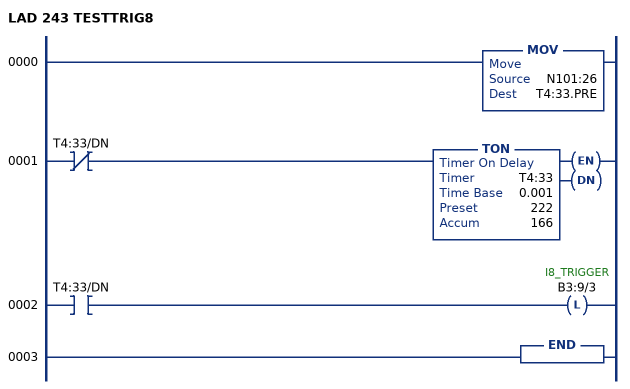
% Rung: 0 %
SOR MOV N101:26 T4:33.PRE EOR
%   N101:26  I8_TRIGTIME %
% Rung: 1 %
SOR XIO T4:33/DN TON T4:33 0.001 222 166 EOR
% Rung: 2 %
SOR XIC T4:33/DN OTL B3:9/3 EOR
%   B3:9/3  I8_TRIGGER %
% Rung: 3 %
SOR END EOR

LADDER 244 "PACKAGER"    % normal %
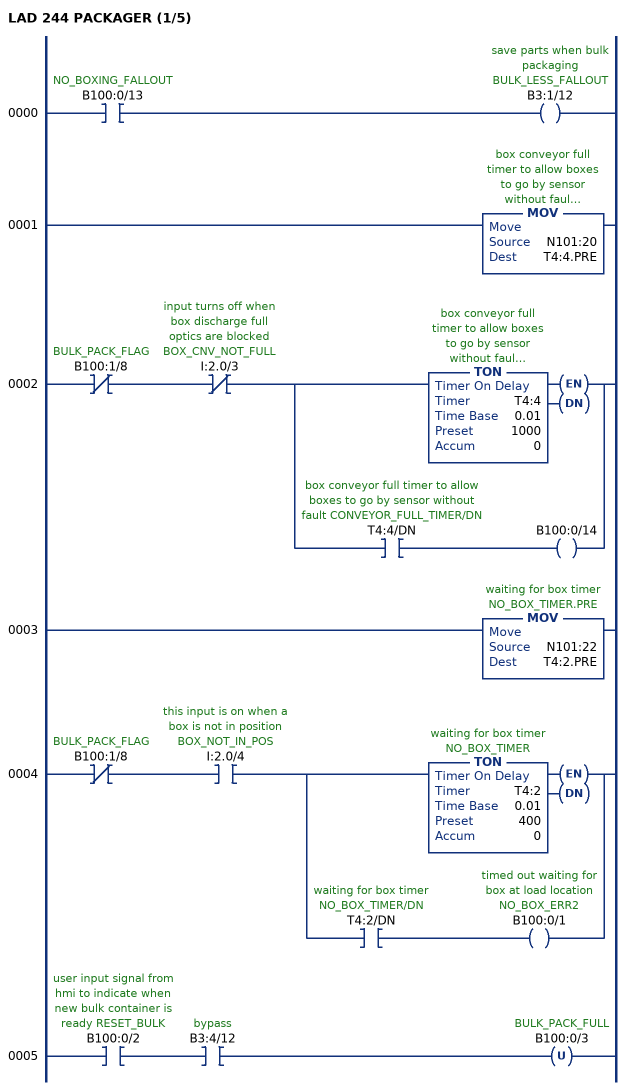
% Rung: 0 %
SOR XIC B100:0/13 OTE B3:1/12 EOR
%   B100:0/13  NO_BOXING_FALLOUT %
%   B3:1/12  BULK_LESS_FALLOUT  "save parts when bulk packaging" %
% Rung: 1 %
SOR MOV N101:20 T4:4.PRE EOR
%   N101:20  CONV_FULL_TIME_LIMIT  "time to allow box to pass box conveyor full sensor without fault" %
%   T4:4  CONVEYOR_FULL_TIMER  "box conveyor full timer to allow boxes to go by sensor without fault" %
% Rung: 2 %
SOR XIO B100:1/8 XIO I:2.0/3 BST TON T4:4 0.01 1000 0 NXB XIC T4:4/DN OTE B100:0/14 BND EOR
%   B100:1/8  BULK_PACK_FLAG %
%   I:2.0/3  BOX_CNV_NOT_FULL  "input turns off when box discharge full optics are blocked" %
%   T4:4  CONVEYOR_FULL_TIMER  "box conveyor full timer to allow boxes to go by sensor without fault" %
% Rung: 3 %
SOR MOV N101:22 T4:2.PRE EOR
%   N101:22  BOX_WAIT_TIME_LIMIT  "the time until waiting for box message in hmi (fault)" %
%   T4:2  NO_BOX_TIMER  "waiting for box timer" %
% Rung: 4 %
SOR XIO B100:1/8 XIC I:2.0/4 BST TON T4:2 0.01 400 0 NXB XIC T4:2/DN OTE B100:0/1 BND EOR
%   B100:1/8  BULK_PACK_FLAG %
%   I:2.0/4  BOX_NOT_IN_POS  "this input is on when a box is not in position" %
%   T4:2  NO_BOX_TIMER  "waiting for box timer" %
%   B100:0/1  NO_BOX_ERR2  "timed out waiting for box at load location" %
% Rung: 5 %
SOR XIC B100:0/2 XIC B3:4/12 OTU B100:0/3 EOR
%   B100:0/2  RESET_BULK  "user input signal from hmi to indicate when new bulk container is ready" %
%   B3:4/12  "bypass" %
%   B100:0/3  BULK_PACK_FULL %

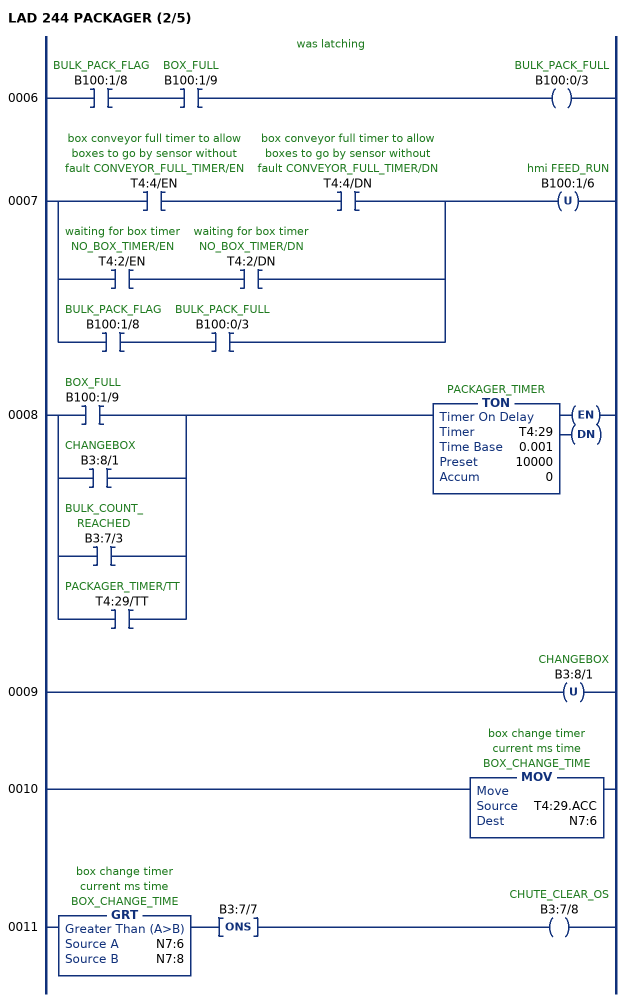
% Rung: 6 %
% was latching %
SOR XIC B100:1/8 XIC B100:1/9 OTE B100:0/3 EOR
%   B100:1/8  BULK_PACK_FLAG %
%   B100:1/9  BOX_FULL %
%   B100:0/3  BULK_PACK_FULL %
% Rung: 7 %
SOR BST XIC T4:4/EN XIC T4:4/DN NXB XIC T4:2/EN XIC T4:2/DN NXB XIC B100:1/8 XIC B100:0/3 BND OTU B100:1/6 EOR
%   T4:4  CONVEYOR_FULL_TIMER  "box conveyor full timer to allow boxes to go by sensor without fault" %
%   T4:2  NO_BOX_TIMER  "waiting for box timer" %
%   B100:1/8  BULK_PACK_FLAG %
%   B100:0/3  BULK_PACK_FULL %
%   B100:1/6  FEED_RUN  "hmi" %
% Rung: 8 %
SOR BST XIC B100:1/9 NXB XIC B3:8/1 NXB XIC B3:7/3 NXB XIC T4:29/TT BND TON T4:29 0.001 10000 0 EOR
%   B100:1/9  BOX_FULL %
%   B3:8/1  CHANGEBOX %
%   B3:7/3  BULK_COUNT_REACHED %
%   T4:29  PACKAGER_TIMER %
% Rung: 9 %
SOR OTU B3:8/1 EOR
%   B3:8/1  CHANGEBOX %
% Rung: 10 %
SOR MOV T4:29.ACC N7:6 EOR
%   T4:29  PACKAGER_TIMER %
%   N7:6  BOX_CHANGE_TIME  "box change timer current ms time" %
% Rung: 11 %
SOR GRT N7:6 N7:8 ONS B3:7/7 OTE B3:7/8 EOR
%   N7:6  BOX_CHANGE_TIME  "box change timer current ms time" %
%   N7:8  CHUTE_CLEAR_TIME %
%   B3:7/8  CHUTE_CLEAR_OS %

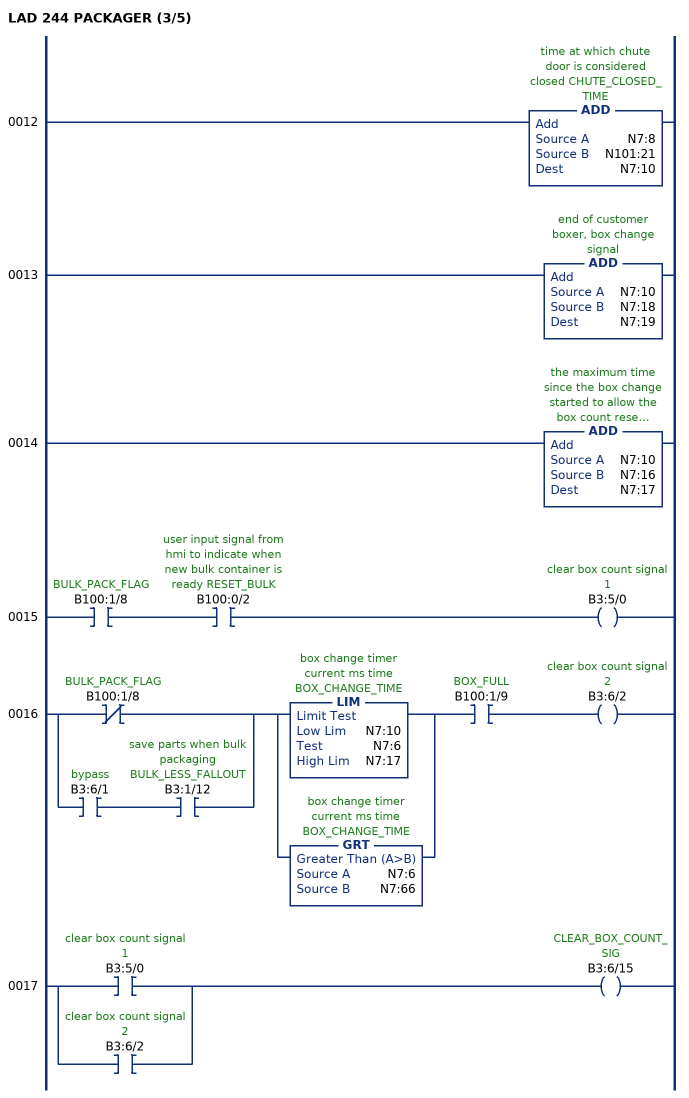
% Rung: 12 %
SOR ADD N7:8 N101:21 N7:10 EOR
%   N7:8  CHUTE_CLEAR_TIME %
%   N101:21  CHUTE_CLOSE_TIME  "ms time required to close chute" %
%   N7:10  CHUTE_CLOSED_TIME  "time at which chute door is considered closed" %
% Rung: 13 %
SOR ADD N7:10 N7:18 N7:19 EOR
%   N7:10  CHUTE_CLOSED_TIME  "time at which chute door is considered closed" %
%   N7:18  CHANGE_BOX_SIG_TIME  "customer boxer change box signal time" %
%   N7:19  "end of customer boxer, box change signal" %
% Rung: 14 %
SOR ADD N7:10 N7:16 N7:17 EOR
%   N7:10  CHUTE_CLOSED_TIME  "time at which chute door is considered closed" %
%   N7:16  RESET_COUNT_SIG_TIME  "maximum length of time to hold box count reset signal on" %
%   N7:17  "the maximum time since the box change started to allow the box count reset signal" %
% Rung: 15 %
SOR XIC B100:1/8 XIC B100:0/2 OTE B3:5/0 EOR
%   B100:1/8  BULK_PACK_FLAG %
%   B100:0/2  RESET_BULK  "user input signal from hmi to indicate when new bulk container is ready" %
%   B3:5/0  "clear box count signal 1" %
% Rung: 16 %
SOR BST XIO B100:1/8 NXB XIC B3:6/1 XIC B3:1/12 BND BST LIM N7:10 N7:6 N7:17 NXB GRT N7:6 N7:66 BND XIC B100:1/9 OTE B3:6/2 EOR
%   B100:1/8  BULK_PACK_FLAG %
%   B3:6/1  "bypass" %
%   B3:1/12  BULK_LESS_FALLOUT  "save parts when bulk packaging" %
%   N7:10  CHUTE_CLOSED_TIME  "time at which chute door is considered closed" %
%   N7:6  BOX_CHANGE_TIME  "box change timer current ms time" %
%   N7:17  "the maximum time since the box change started to allow the box count reset signal" %
%   B100:1/9  BOX_FULL %
%   B3:6/2  "clear box count signal 2" %
% Rung: 17 %
SOR BST XIC B3:5/0 NXB XIC B3:6/2 BND OTE B3:6/15 EOR
%   B3:5/0  "clear box count signal 1" %
%   B3:6/2  "clear box count signal 2" %
%   B3:6/15  CLEAR_BOX_COUNT_SIG %

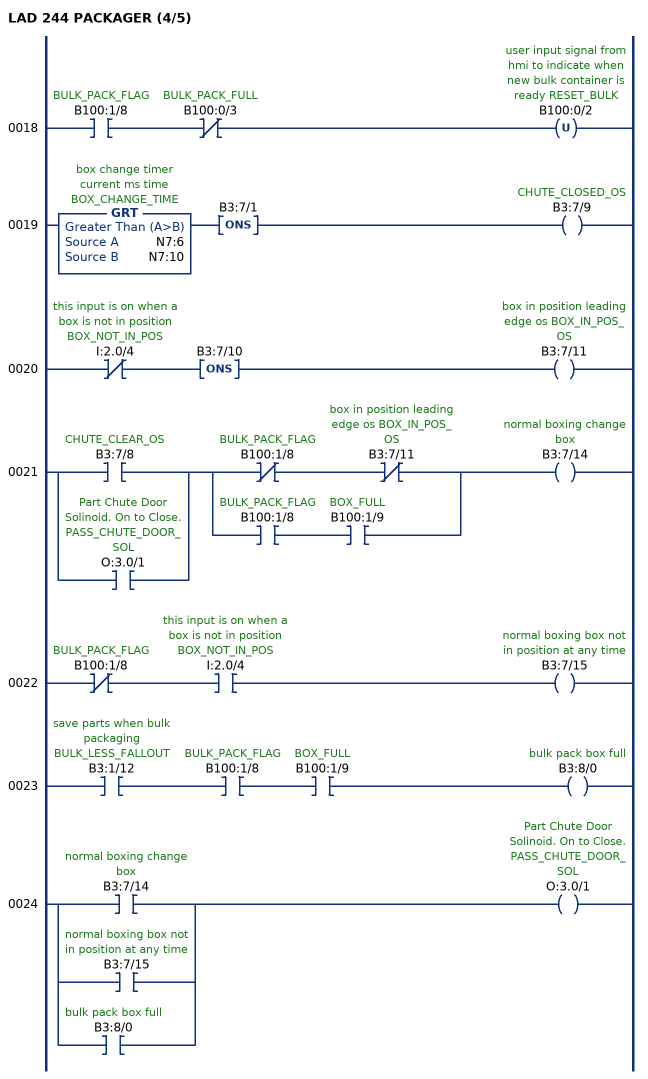
% Rung: 18 %
SOR XIC B100:1/8 XIO B100:0/3 OTU B100:0/2 EOR
%   B100:1/8  BULK_PACK_FLAG %
%   B100:0/3  BULK_PACK_FULL %
%   B100:0/2  RESET_BULK  "user input signal from hmi to indicate when new bulk container is ready" %
% Rung: 19 %
SOR GRT N7:6 N7:10 ONS B3:7/1 OTE B3:7/9 EOR
%   N7:6  BOX_CHANGE_TIME  "box change timer current ms time" %
%   N7:10  CHUTE_CLOSED_TIME  "time at which chute door is considered closed" %
%   B3:7/9  CHUTE_CLOSED_OS %
% Rung: 20 %
SOR XIO I:2.0/4 ONS B3:7/10 OTE B3:7/11 EOR
%   I:2.0/4  BOX_NOT_IN_POS  "this input is on when a box is not in position" %
%   B3:7/11  BOX_IN_POS_OS  "box in position leading edge os" %
% Rung: 21 %
SOR BST XIC B3:7/8 NXB XIC O:3.0/1 BND BST XIO B100:1/8 XIO B3:7/11 NXB XIC B100:1/8 XIC B100:1/9 BND OTE B3:7/14 EOR
%   B3:7/8  CHUTE_CLEAR_OS %
%   O:3.0/1  PASS_CHUTE_DOOR_SOL  "Part Chute Door Solinoid. On to Close." %
%   B100:1/8  BULK_PACK_FLAG %
%   B3:7/11  BOX_IN_POS_OS  "box in position leading edge os" %
%   B100:1/9  BOX_FULL %
%   B3:7/14  "normal boxing change box" %
% Rung: 22 %
SOR XIO B100:1/8 XIC I:2.0/4 OTE B3:7/15 EOR
%   B100:1/8  BULK_PACK_FLAG %
%   I:2.0/4  BOX_NOT_IN_POS  "this input is on when a box is not in position" %
%   B3:7/15  "normal boxing box not in position at any time" %
% Rung: 23 %
SOR XIC B3:1/12 XIC B100:1/8 XIC B100:1/9 OTE B3:8/0 EOR
%   B3:1/12  BULK_LESS_FALLOUT  "save parts when bulk packaging" %
%   B100:1/8  BULK_PACK_FLAG %
%   B100:1/9  BOX_FULL %
%   B3:8/0  "bulk pack box full" %
% Rung: 24 %
SOR BST XIC B3:7/14 NXB XIC B3:7/15 NXB XIC B3:8/0 BND OTE O:3.0/1 EOR
%   B3:7/14  "normal boxing change box" %
%   B3:7/15  "normal boxing box not in position at any time" %
%   B3:8/0  "bulk pack box full" %
%   O:3.0/1  PASS_CHUTE_DOOR_SOL  "Part Chute Door Solinoid. On to Close." %

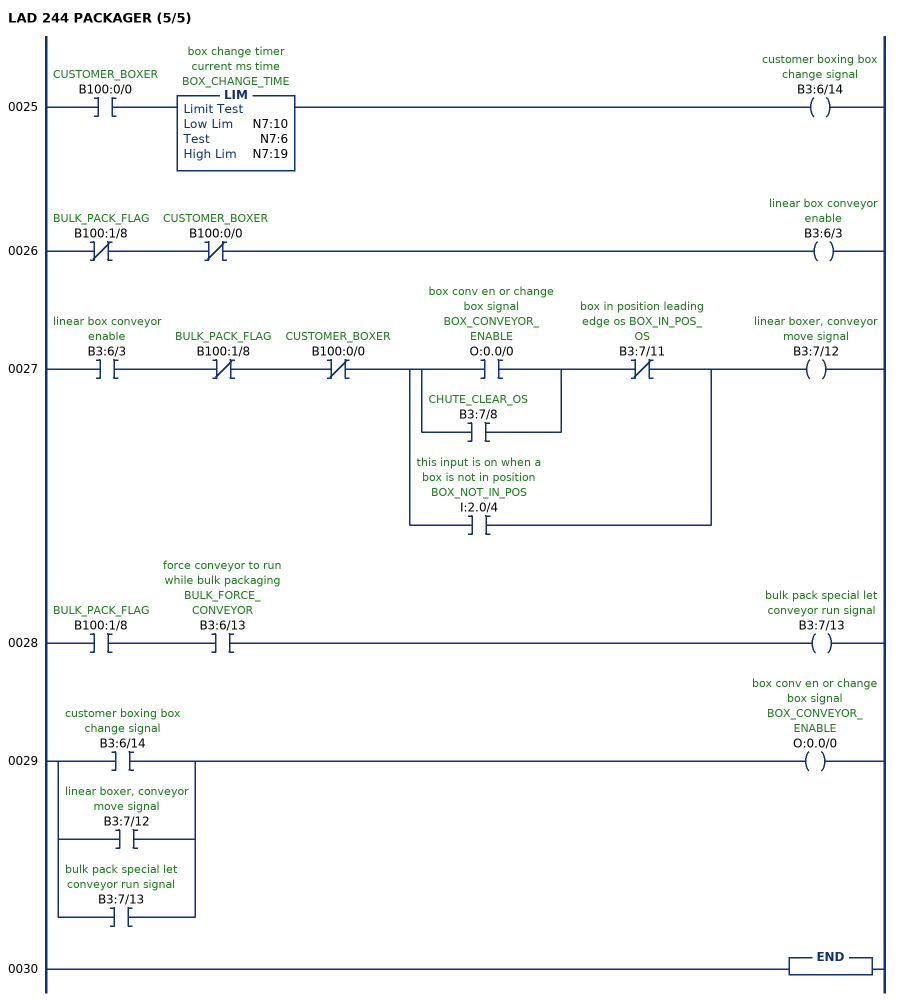
% Rung: 25 %
SOR XIC B100:0/0 LIM N7:10 N7:6 N7:19 OTE B3:6/14 EOR
%   B100:0/0  CUSTOMER_BOXER %
%   N7:10  CHUTE_CLOSED_TIME  "time at which chute door is considered closed" %
%   N7:6  BOX_CHANGE_TIME  "box change timer current ms time" %
%   N7:19  "end of customer boxer, box change signal" %
%   B3:6/14  "customer boxing box change signal" %
% Rung: 26 %
SOR XIO B100:1/8 XIO B100:0/0 OTE B3:6/3 EOR
%   B100:1/8  BULK_PACK_FLAG %
%   B100:0/0  CUSTOMER_BOXER %
%   B3:6/3  "linear box conveyor enable" %
% Rung: 27 %
SOR XIC B3:6/3 XIO B100:1/8 XIO B100:0/0 BST BST XIC O:0.0/0 NXB XIC B3:7/8 BND XIO B3:7/11 NXB XIC I:2.0/4 BND OTE B3:7/12 EOR
%   B3:6/3  "linear box conveyor enable" %
%   B100:1/8  BULK_PACK_FLAG %
%   B100:0/0  CUSTOMER_BOXER %
%   O:0.0/0  BOX_CONVEYOR_ENABLE  "box conv en or change box signal" %
%   B3:7/8  CHUTE_CLEAR_OS %
%   B3:7/11  BOX_IN_POS_OS  "box in position leading edge os" %
%   I:2.0/4  BOX_NOT_IN_POS  "this input is on when a box is not in position" %
%   B3:7/12  "linear boxer, conveyor move signal" %
% Rung: 28 %
SOR XIC B100:1/8 XIC B3:6/13 OTE B3:7/13 EOR
%   B100:1/8  BULK_PACK_FLAG %
%   B3:6/13  BULK_FORCE_CONVEYOR  "force conveyor to run while bulk packaging" %
%   B3:7/13  "bulk pack special let conveyor run signal" %
% Rung: 29 %
SOR BST XIC B3:6/14 NXB XIC B3:7/12 NXB XIC B3:7/13 BND OTE O:0.0/0 EOR
%   B3:6/14  "customer boxing box change signal" %
%   B3:7/12  "linear boxer, conveyor move signal" %
%   B3:7/13  "bulk pack special let conveyor run signal" %
%   O:0.0/0  BOX_CONVEYOR_ENABLE  "box conv en or change box signal" %
% Rung: 30 %
SOR END EOR

LADDER 245 "NO PACKAGE"
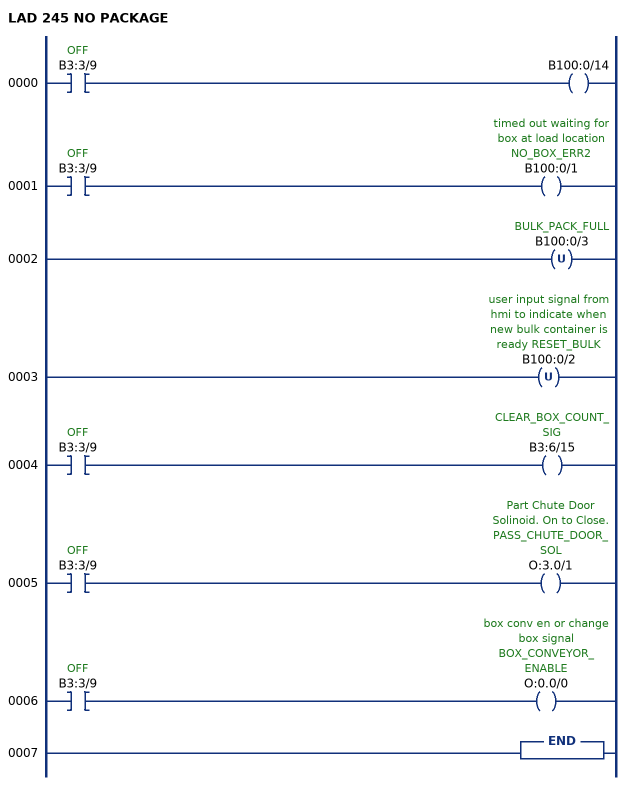
% Rung: 0 %
SOR XIC B3:3/9 OTE B100:0/14 EOR
%   B3:3/9  OFF %
% Rung: 1 %
SOR XIC B3:3/9 OTE B100:0/1 EOR
%   B3:3/9  OFF %
%   B100:0/1  NO_BOX_ERR2  "timed out waiting for box at load location" %
% Rung: 2 %
SOR OTU B100:0/3 EOR
%   B100:0/3  BULK_PACK_FULL %
% Rung: 3 %
SOR OTU B100:0/2 EOR
%   B100:0/2  RESET_BULK  "user input signal from hmi to indicate when new bulk container is ready" %
% Rung: 4 %
SOR XIC B3:3/9 OTE B3:6/15 EOR
%   B3:3/9  OFF %
%   B3:6/15  CLEAR_BOX_COUNT_SIG %
% Rung: 5 %
SOR XIC B3:3/9 OTE O:3.0/1 EOR
%   B3:3/9  OFF %
%   O:3.0/1  PASS_CHUTE_DOOR_SOL  "Part Chute Door Solinoid. On to Close." %
% Rung: 6 %
SOR XIC B3:3/9 OTE O:0.0/0 EOR
%   B3:3/9  OFF %
%   O:0.0/0  BOX_CONVEYOR_ENABLE  "box conv en or change box signal" %
% Rung: 7 %
SOR END EOR

LADDER 246 "RATE1"
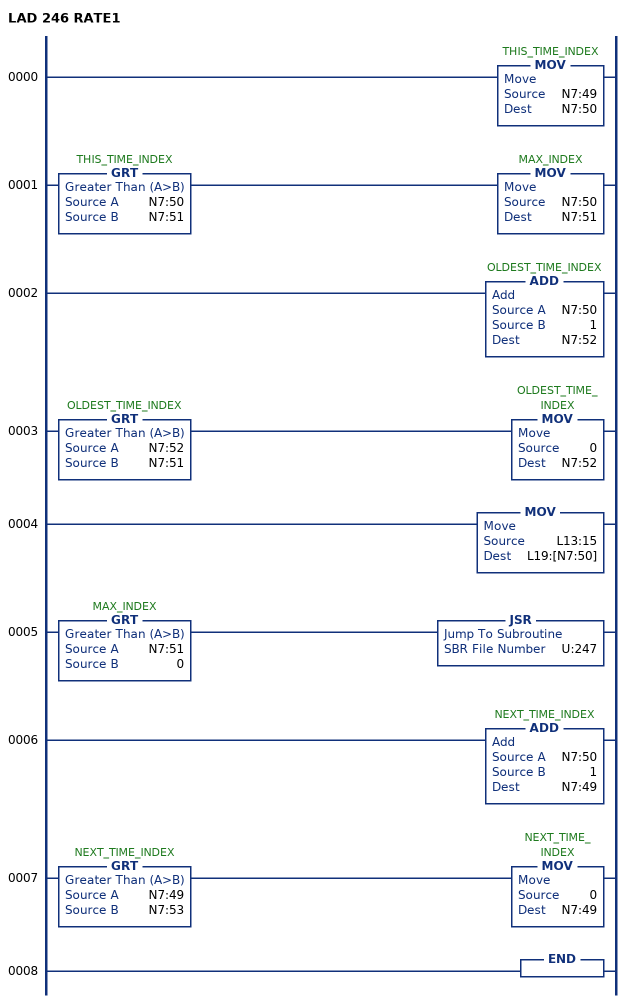
% Rung: 0 %
SOR MOV N7:49 N7:50 EOR
%   N7:49  NEXT_TIME_INDEX %
%   N7:50  THIS_TIME_INDEX %
% Rung: 1 %
SOR GRT N7:50 N7:51 MOV N7:50 N7:51 EOR
%   N7:50  THIS_TIME_INDEX %
%   N7:51  MAX_INDEX %
% Rung: 2 %
SOR ADD N7:50 1 N7:52 EOR
%   N7:50  THIS_TIME_INDEX %
%   N7:52  OLDEST_TIME_INDEX %
% Rung: 3 %
SOR GRT N7:52 N7:51 MOV 0 N7:52 EOR
%   N7:52  OLDEST_TIME_INDEX %
%   N7:51  MAX_INDEX %
% Rung: 4 %
SOR MOV L13:15 L19:[N7:50] EOR
%   L13:15  THE_TIME %
%   N7:50  THIS_TIME_INDEX %
% Rung: 5 %
SOR GRT N7:51 0 JSR U:247 EOR
%   N7:51  MAX_INDEX %
% Rung: 6 %
SOR ADD N7:50 1 N7:49 EOR
%   N7:50  THIS_TIME_INDEX %
%   N7:49  NEXT_TIME_INDEX %
% Rung: 7 %
SOR GRT N7:49 N7:53 MOV 0 N7:49 EOR
%   N7:49  NEXT_TIME_INDEX %
%   N7:53  UPPER_INDEX_LIMIT %
% Rung: 8 %
SOR END EOR

LADDER 247 "RATE2"
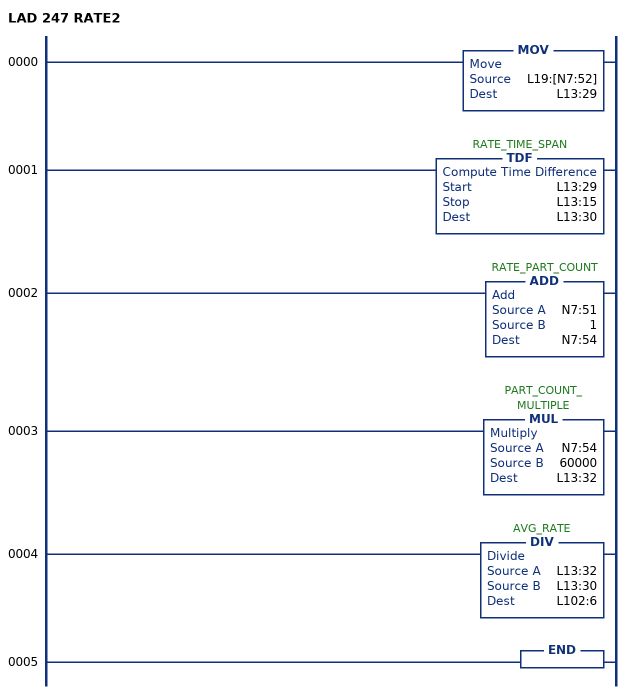
% Rung: 0 %
SOR MOV L19:[N7:52] L13:29 EOR
%   N7:52  OLDEST_TIME_INDEX %
% Rung: 1 %
SOR TDF L13:29 L13:15 L13:30 EOR
%   L13:15  THE_TIME %
%   L13:30  RATE_TIME_SPAN %
% Rung: 2 %
SOR ADD N7:51 1 N7:54 EOR
%   N7:51  MAX_INDEX %
%   N7:54  RATE_PART_COUNT %
% Rung: 3 %
SOR MUL N7:54 60000 L13:32 EOR
%   N7:54  RATE_PART_COUNT %
%   L13:32  PART_COUNT_MULTIPLE %
% Rung: 4 %
SOR DIV L13:32 L13:30 L102:6 EOR
%   L13:32  PART_COUNT_MULTIPLE %
%   L13:30  RATE_TIME_SPAN %
%   L102:6  AVG_RATE %
% Rung: 5 %
SOR END EOR

LADDER 248 "RESET RATE"
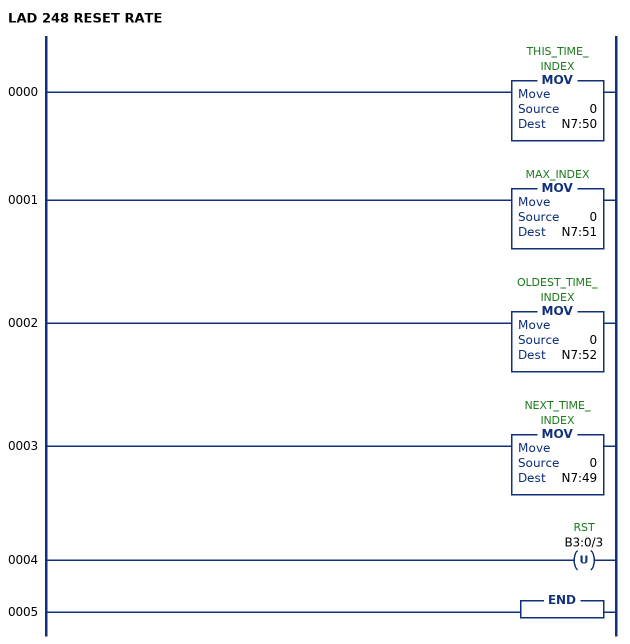
% Rung: 0 %
SOR MOV 0 N7:50 EOR
%   N7:50  THIS_TIME_INDEX %
% Rung: 1 %
SOR MOV 0 N7:51 EOR
%   N7:51  MAX_INDEX %
% Rung: 2 %
SOR MOV 0 N7:52 EOR
%   N7:52  OLDEST_TIME_INDEX %
% Rung: 3 %
SOR MOV 0 N7:49 EOR
%   N7:49  NEXT_TIME_INDEX %
% Rung: 4 %
SOR OTU B3:0/3 EOR
%   B3:0/3  RST %
% Rung: 5 %
SOR END EOR

LADDER 249 "NP STOP"    % stop on no good %
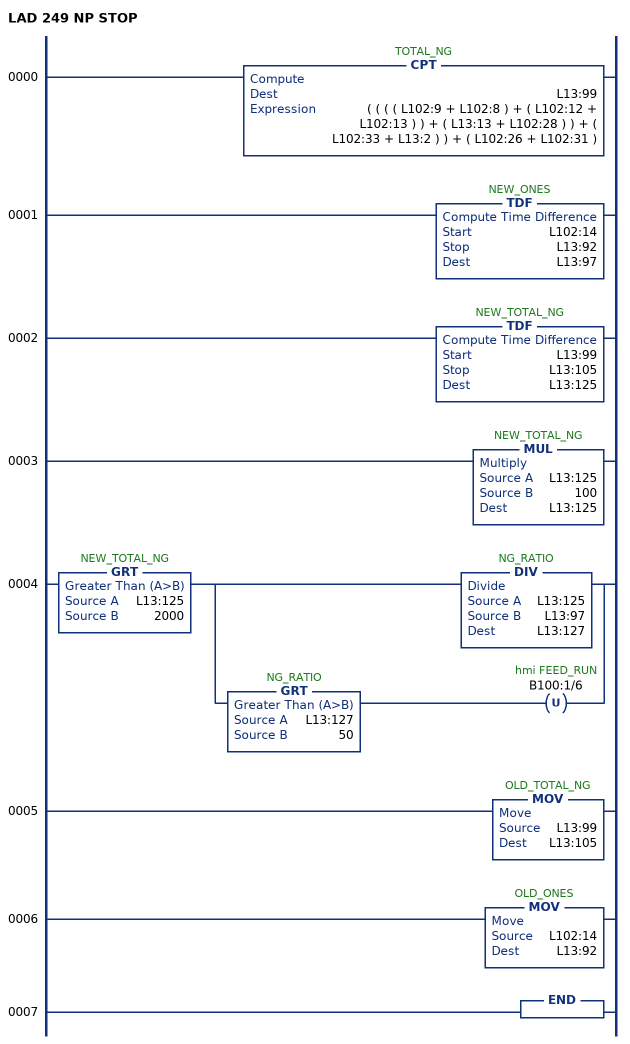
% Rung: 0 %
SOR CPT L13:99 " ( ( ( ( L102:9 + L102:8 ) + ( L102:12 + L102:13 ) ) + ( L13:13 + L102:28 ) ) + ( L102:33 + L13:2 ) ) + ( L102:26 + L102:31 ) " EOR
%   L13:99  TOTAL_NG %
%   L102:9  "too wide bottom" %
%   L102:8  "too close bottom" %
%   L102:12  "too close top count" %
%   L102:13  "too wide top count" %
%   L102:28  I1_I5_SKIPPEDCOUNT %
%   L102:33  I2_I6_SKIPPEDCOUNT %
%   L102:26  I1_I5_FAIL_COUNT %
%   L102:31  I2_I6_FAIL_COUNT %
% Rung: 1 %
SOR TDF L102:14 L13:92 L13:97 EOR
%   L102:14  ONES %
%   L13:92  OLD_ONES %
%   L13:97  NEW_ONES %
% Rung: 2 %
SOR TDF L13:99 L13:105 L13:125 EOR
%   L13:99  TOTAL_NG %
%   L13:105  OLD_TOTAL_NG %
%   L13:125  NEW_TOTAL_NG %
% Rung: 3 %
SOR MUL L13:125 100 L13:125 EOR
%   L13:125  NEW_TOTAL_NG %
% Rung: 4 %
SOR GRT L13:125 2000 BST DIV L13:125 L13:97 L13:127 NXB GRT L13:127 50 OTU B100:1/6 BND EOR
%   L13:125  NEW_TOTAL_NG %
%   L13:97  NEW_ONES %
%   L13:127  NG_RATIO %
%   B100:1/6  FEED_RUN  "hmi" %
% Rung: 5 %
SOR MOV L13:99 L13:105 EOR
%   L13:99  TOTAL_NG %
%   L13:105  OLD_TOTAL_NG %
% Rung: 6 %
SOR MOV L102:14 L13:92 EOR
%   L102:14  ONES %
%   L13:92  OLD_ONES %
% Rung: 7 %
SOR END EOR

LADDER 250 "SPEED BOT"    % high speed %
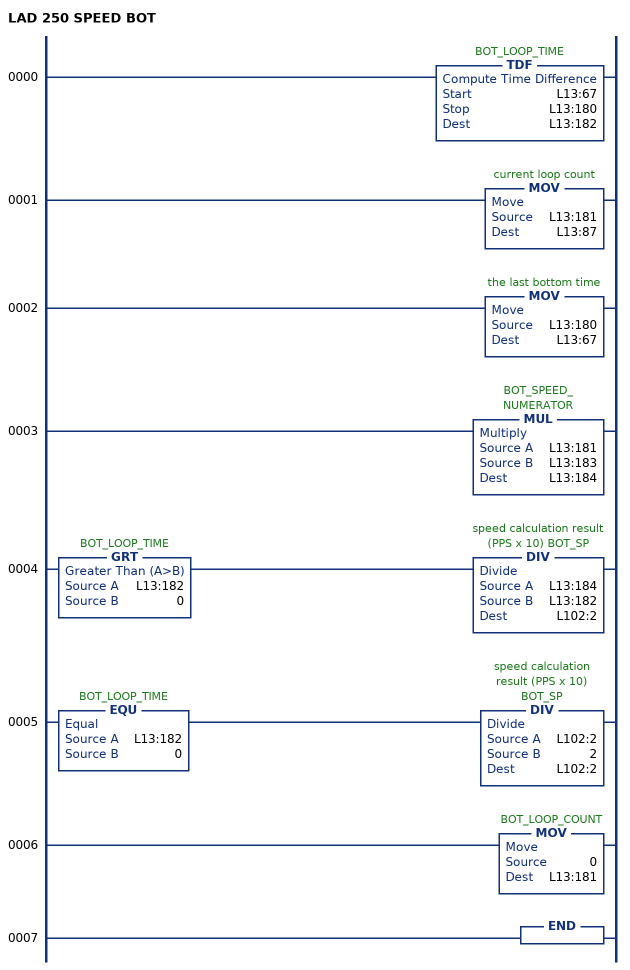
% Rung: 0 %
SOR TDF L13:67 L13:180 L13:182 EOR
%   L13:67  "the last bottom time" %
%   L13:180  BOT_THIS_TIME  "rtc bot belt movement event time" %
%   L13:182  BOT_LOOP_TIME %
% Rung: 1 %
SOR MOV L13:181 L13:87 EOR
%   L13:181  BOT_LOOP_COUNT %
%   L13:87  "current loop count" %
% Rung: 2 %
SOR MOV L13:180 L13:67 EOR
%   L13:180  BOT_THIS_TIME  "rtc bot belt movement event time" %
%   L13:67  "the last bottom time" %
% Rung: 3 %
SOR MUL L13:181 L13:183 L13:184 EOR
%   L13:181  BOT_LOOP_COUNT %
%   L13:183  TKS_PER_SECOND %
%   L13:184  BOT_SPEED_NUMERATOR %
% Rung: 4 %
SOR GRT L13:182 0 DIV L13:184 L13:182 L102:2 EOR
%   L13:182  BOT_LOOP_TIME %
%   L13:184  BOT_SPEED_NUMERATOR %
%   L102:2  BOT_SP  "speed calculation result (PPS x 10)" %
% Rung: 5 %
SOR EQU L13:182 0 DIV L102:2 2 L102:2 EOR
%   L13:182  BOT_LOOP_TIME %
%   L102:2  BOT_SP  "speed calculation result (PPS x 10)" %
% Rung: 6 %
SOR MOV 0 L13:181 EOR
%   L13:181  BOT_LOOP_COUNT %
% Rung: 7 %
SOR END EOR

LADDER 251 "SPEED TOP"    % high speed %
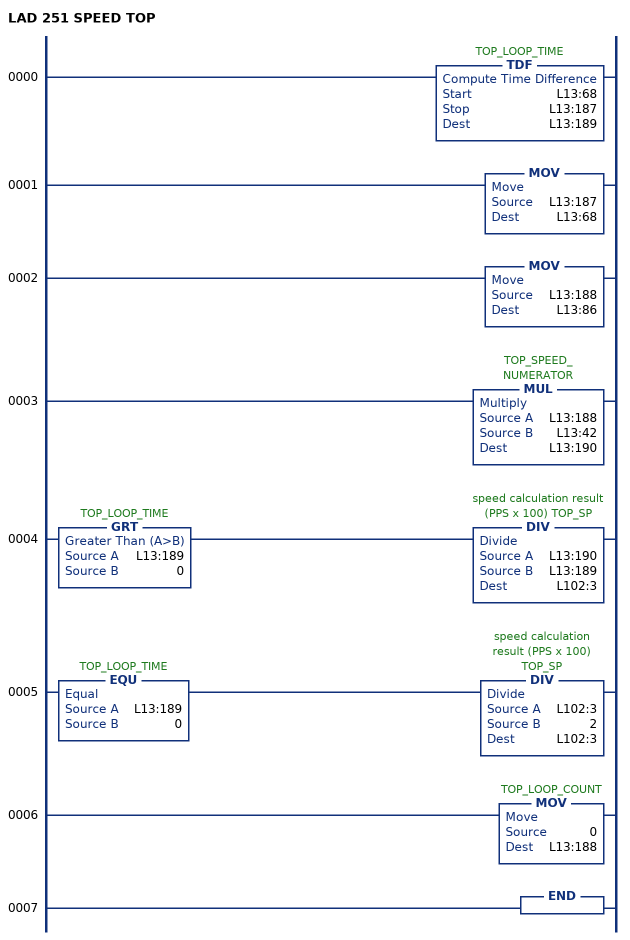
% Rung: 0 %
SOR TDF L13:68 L13:187 L13:189 EOR
%   L13:187  TOP_THIS_TIME  "rtc top belt movement event time" %
%   L13:189  TOP_LOOP_TIME %
% Rung: 1 %
SOR MOV L13:187 L13:68 EOR
%   L13:187  TOP_THIS_TIME  "rtc top belt movement event time" %
% Rung: 2 %
SOR MOV L13:188 L13:86 EOR
%   L13:188  TOP_LOOP_COUNT %
% Rung: 3 %
SOR MUL L13:188 L13:42 L13:190 EOR
%   L13:188  TOP_LOOP_COUNT %
%   L13:190  TOP_SPEED_NUMERATOR %
% Rung: 4 %
SOR GRT L13:189 0 DIV L13:190 L13:189 L102:3 EOR
%   L13:189  TOP_LOOP_TIME %
%   L13:190  TOP_SPEED_NUMERATOR %
%   L102:3  TOP_SP  "speed calculation result (PPS x 100)" %
% Rung: 5 %
SOR EQU L13:189 0 DIV L102:3 2 L102:3 EOR
%   L13:189  TOP_LOOP_TIME %
%   L102:3  TOP_SP  "speed calculation result (PPS x 100)" %
% Rung: 6 %
SOR MOV 0 L13:188 EOR
%   L13:188  TOP_LOOP_COUNT %
% Rung: 7 %
SOR END EOR

LADDER 252 "P BOT"    % high speed %
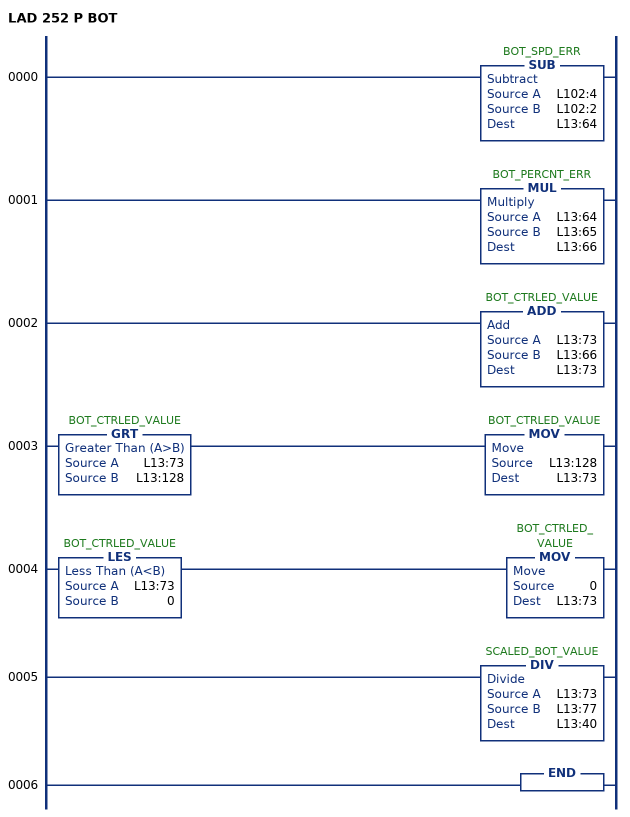
% Rung: 0 %
SOR SUB L102:4 L102:2 L13:64 EOR
%   L102:4  BOT_SPD_SETPOINT %
%   L102:2  BOT_SP  "speed calculation result (PPS x 10)" %
%   L13:64  BOT_SPD_ERR %
% Rung: 1 %
SOR MUL L13:64 L13:65 L13:66 EOR
%   L13:64  BOT_SPD_ERR %
%   L13:65  POS5SHIFT %
%   L13:66  BOT_PERCNT_ERR %
% Rung: 2 %
SOR ADD L13:73 L13:66 L13:73 EOR
%   L13:73  BOT_CTRLED_VALUE %
%   L13:66  BOT_PERCNT_ERR %
% Rung: 3 %
SOR GRT L13:73 L13:128 MOV L13:128 L13:73 EOR
%   L13:73  BOT_CTRLED_VALUE %
%   L13:128  "how much top has shifted since measurment" %
% Rung: 4 %
SOR LES L13:73 0 MOV 0 L13:73 EOR
%   L13:73  BOT_CTRLED_VALUE %
% Rung: 5 %
SOR DIV L13:73 L13:77 L13:40 EOR
%   L13:73  BOT_CTRLED_VALUE %
%   L13:40  SCALED_BOT_VALUE %
% Rung: 6 %
SOR END EOR

LADDER 253 "P TOP"    % high speed %
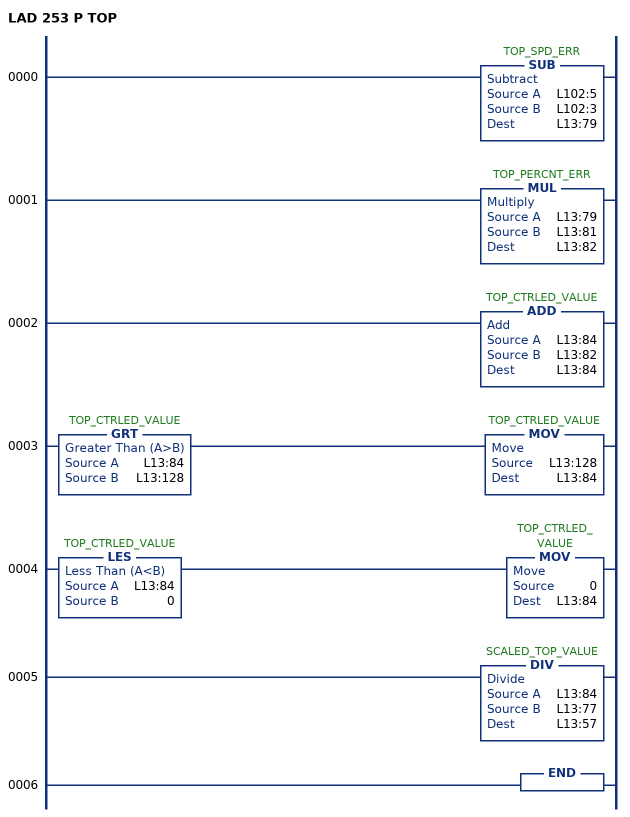
% Rung: 0 %
SOR SUB L102:5 L102:3 L13:79 EOR
%   L102:5  TOP_SPD_SETPOINT %
%   L102:3  TOP_SP  "speed calculation result (PPS x 100)" %
%   L13:79  TOP_SPD_ERR %
% Rung: 1 %
SOR MUL L13:79 L13:81 L13:82 EOR
%   L13:79  TOP_SPD_ERR %
%   L13:81  TOP_FDBK_RATIO %
%   L13:82  TOP_PERCNT_ERR %
% Rung: 2 %
SOR ADD L13:84 L13:82 L13:84 EOR
%   L13:84  TOP_CTRLED_VALUE %
%   L13:82  TOP_PERCNT_ERR %
% Rung: 3 %
SOR GRT L13:84 L13:128 MOV L13:128 L13:84 EOR
%   L13:84  TOP_CTRLED_VALUE %
%   L13:128  "how much top has shifted since measurment" %
% Rung: 4 %
SOR LES L13:84 0 MOV 0 L13:84 EOR
%   L13:84  TOP_CTRLED_VALUE %
% Rung: 5 %
SOR DIV L13:84 L13:77 L13:57 EOR
%   L13:84  TOP_CTRLED_VALUE %
%   L13:57  SCALED_TOP_VALUE %
% Rung: 6 %
SOR END EOR

LADDER 254 "TOTALCOUNT"
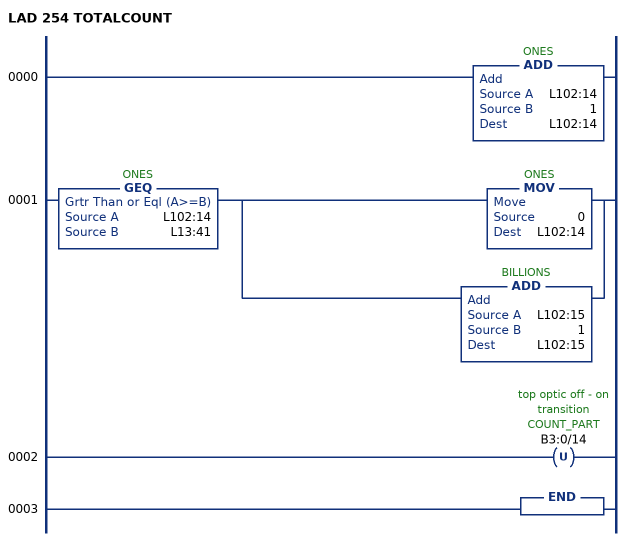
% Rung: 0 %
SOR ADD L102:14 1 L102:14 EOR
%   L102:14  ONES %
% Rung: 1 %
SOR GEQ L102:14 L13:41 BST MOV 0 L102:14 NXB ADD L102:15 1 L102:15 BND EOR
%   L102:14  ONES %
%   L13:41  "skipped count change in the last 3 seconds" %
%   L102:15  BILLIONS %
% Rung: 2 %
SOR OTU B3:0/14 EOR
%   B3:0/14  COUNT_PART  "top optic off - on transition" %
% Rung: 3 %
SOR END EOR

LADDER 255 "SAVED"
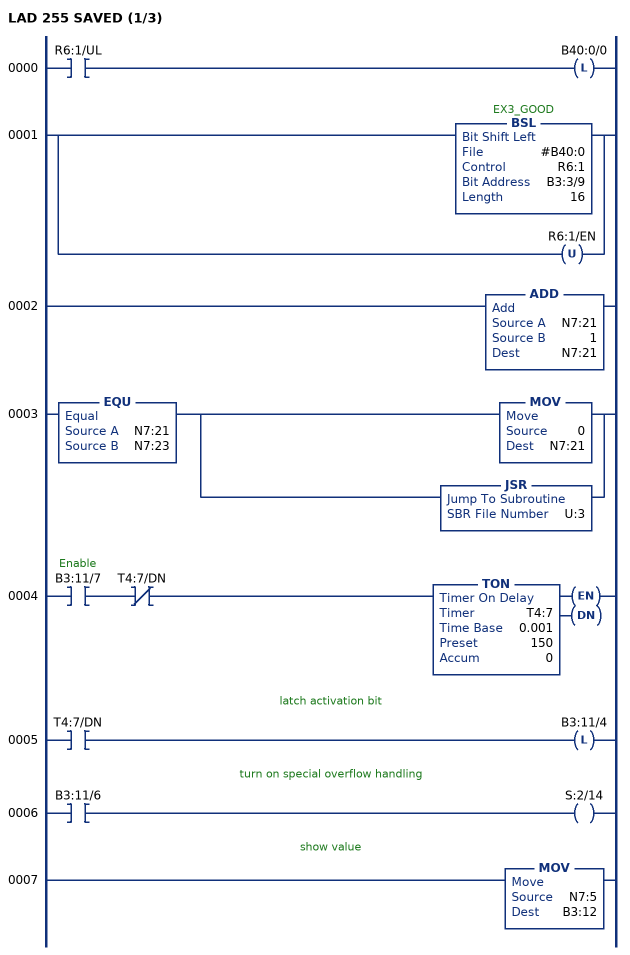
% Rung: 0 %
SOR XIC R6:1/UL OTL B40:0/0 EOR
% Rung: 1 %
SOR BST BSL #B40:0 R6:1 B3:3/9 16 NXB OTU R6:1/EN BND EOR
%   B40:0  EX3_GOOD %
%   B3:3/9  OFF %
% Rung: 2 %
SOR ADD N7:21 1 N7:21 EOR
% Rung: 3 %
SOR EQU N7:21 N7:23 BST MOV 0 N7:21 NXB JSR U:3 BND EOR
% Rung: 4 %
SOR XIC B3:11/7 XIO T4:7/DN TON T4:7 0.001 150 0 EOR
%   B3:11/7  "Enable" %
% Rung: 5 %
% latch activation bit %
SOR XIC T4:7/DN OTL B3:11/4 EOR
% Rung: 6 %
% turn on special overflow handling %
SOR XIC B3:11/6 OTE S:2/14 EOR
% Rung: 7 %
% show value %
SOR MOV N7:5 B3:12 EOR

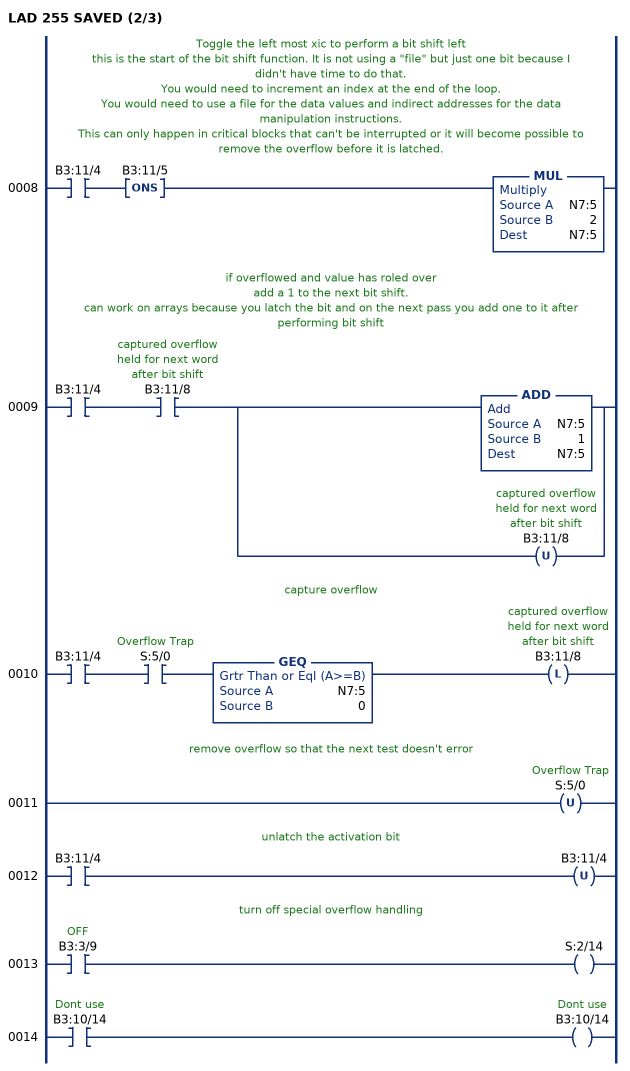
% Rung: 8 %
% Toggle the left most xic to perform a bit shift left
% 
% this is the start of the bit shift function. It is not using a "file" but just one bit because I didn't have time to do that.
% You would need to increment an index at the end of the loop.
% You would need to use a file for the data values and indirect addresses for the data manipulation instructions.
% 
% This can only happen in critical blocks that can't be interrupted or it will become possible to remove the overflow before it is latched. %
SOR XIC B3:11/4 ONS B3:11/5 MUL N7:5 2 N7:5 EOR
% Rung: 9 %
% if overflowed and value has roled over
% add a 1 to the next bit shift.
% can work on arrays because you latch the bit and on the next pass you add one to it after performing bit shift %
SOR XIC B3:11/4 XIC B3:11/8 BST ADD N7:5 1 N7:5 NXB OTU B3:11/8 BND EOR
%   B3:11/8  "captured overflow held for next word after bit shift" %
% Rung: 10 %
% capture overflow %
SOR XIC B3:11/4 XIC S:5/0 GEQ N7:5 0 OTL B3:11/8 EOR
%   S:5/0  "Overflow Trap" %
%   B3:11/8  "captured overflow held for next word after bit shift" %
% Rung: 11 %
% remove overflow so that the next test doesn't error %
SOR OTU S:5/0 EOR
%   S:5/0  "Overflow Trap" %
% Rung: 12 %
% unlatch the activation bit %
SOR XIC B3:11/4 OTU B3:11/4 EOR
% Rung: 13 %
% turn off special overflow handling %
SOR XIC B3:3/9 OTE S:2/14 EOR
%   B3:3/9  OFF %
% Rung: 14 %
SOR XIC B3:10/14 OTE B3:10/14 EOR
%   B3:10/14  "Dont use" %

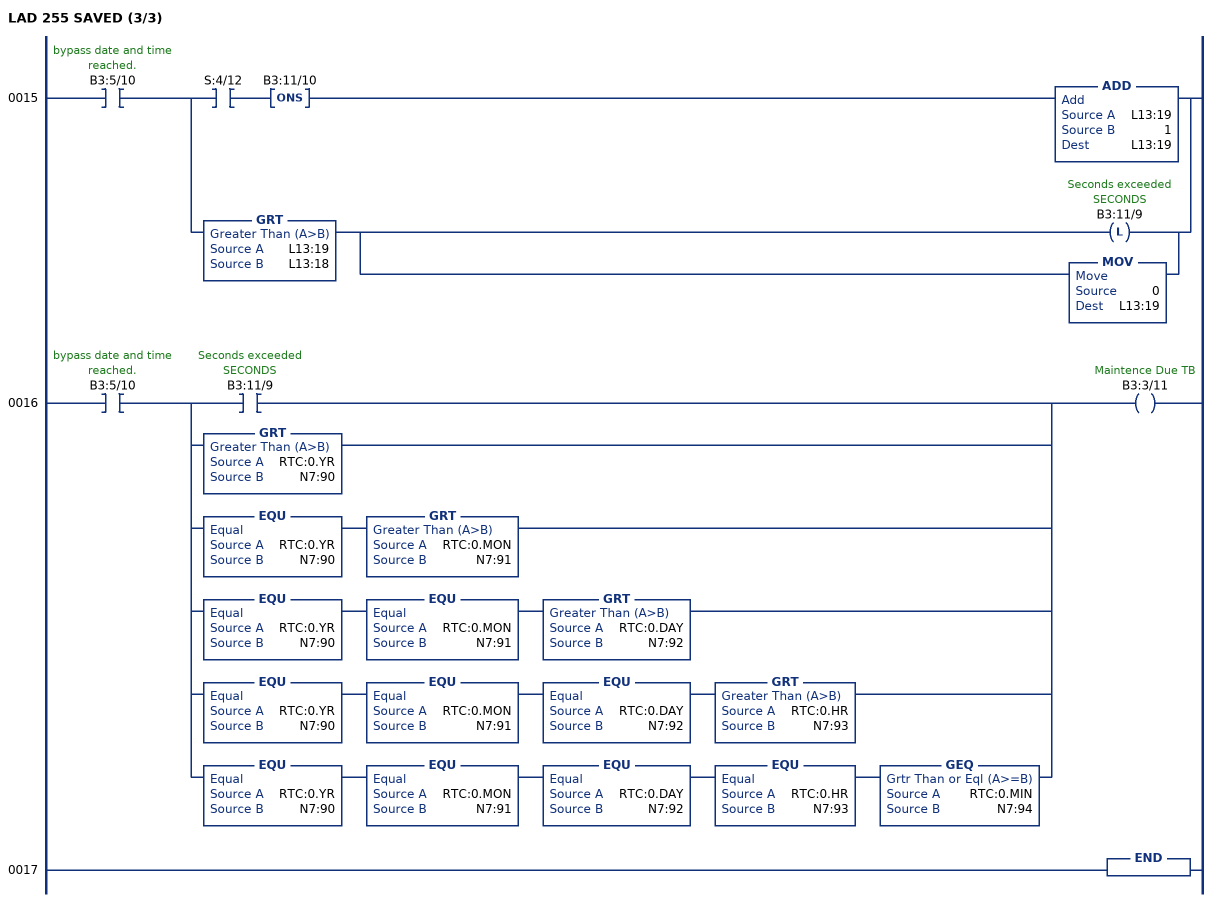
% Rung: 15 %
SOR XIC B3:5/10 BST XIC S:4/12 ONS B3:11/10 ADD L13:19 1 L13:19 NXB GRT L13:19 L13:18 BST OTL B3:11/9 NXB MOV 0 L13:19 BND BND EOR
%   B3:5/10  "bypass date and time reached." %
%   L13:18  MAX %
%   B3:11/9  SECONDS  "Seconds exceeded" %
% Rung: 16 %
SOR XIC B3:5/10 BST XIC B3:11/9 NXB GRT RTC:0.YR N7:90 NXB EQU RTC:0.YR N7:90 GRT RTC:0.MON N7:91 NXB EQU RTC:0.YR N7:90 EQU RTC:0.MON N7:91 GRT RTC:0.DAY N7:92 NXB EQU RTC:0.YR N7:90 EQU RTC:0.MON N7:91 EQU RTC:0.DAY N7:92 GRT RTC:0.HR N7:93 NXB EQU RTC:0.YR N7:90 EQU RTC:0.MON N7:91 EQU RTC:0.DAY N7:92 EQU RTC:0.HR N7:93 GEQ RTC:0.MIN N7:94 BND OTE B3:3/11 EOR
%   B3:5/10  "bypass date and time reached." %
%   B3:11/9  SECONDS  "Seconds exceeded" %
%   N7:90  RTC %
%   B3:3/11  TB  "Maintence Due" %
% Rung: 17 %
SOR END EOR

OTHER DOCUMENTED ADDRESSES
  B189:0/0  "change box"
  B189:0/9  "override boxing ok or not full signal"
  B189:0/11  "HMI force door close"
  B196:1/0  "Chute door is closed"
  B196:1/1  "control chute door"
  B196:1/13  "force box conveyor on"
  B196:3/0  "for hmi to continue production unlatched by hmi"
  HSC:0.0  "top"
  HSC:0.3/6  "Underflow interrupt"
  HSC:0.3/7  "Overflow interrupt"
  HSC:1.0  "bot"
  HSC:1.3/6  "Underflow interrupt"
  HSC:1.3/7  "Overflow interrupt"
  I7_TRAC  
  I:0.0/0  "Encoder Signal "A""
  I:0.0/1  "Encoder Signal "B""
  I:0.0/4  "Encoder Signal "A""
  I:0.0/5  "Encoder Signal "B""
  I:0.1/4  "not used"
  I:0.1/5  "not used"
  I:0.1/6  "not used"
  I:0.1/7  "not used"
  I:0.1/8  "not used"
  I:0.1/9  "not used"
  I:0.1/10  "not used"
  I:0.1/11  "not used"
  I:0.1/12  "not used"
  I:0.1/13  "not used"
  I:0.1/14  "not used"
  I:0.1/15  "not used"
  I:0.2  "not used"
  I:0.2/3  "Packaging Conveyor full"
  I:0.2/4  "Packaging Conveyor Box in Position"
  I:0.3  "not used"
  I:0.4  "Spare Analog Input 1"
  I:0.5  "Spare Analog Input 2"
  I:0.6  "Spare Analog Input 3"
  I:2.0/0  FRONT_ESTOP
  I:2.0/1  REAR_ESTOP
  I:2.0/8  FRONT_DOOR  "front door signal ce models only"
  I:2.0/9  REAR_DOOR  "rear door signal ce models only"
  I:2.0/11  "spare"
  L23:19  TOP_OPT_FAIL_CT
  L23:34  AIR_PRESSURE_FAULT
  L28:0  INS_1_TIME
  L29:0  INS_1_POS
  L30:0  INS_5_TIME
  L31:0  INS_5_POS
  L32:0  INS_6_TIME
  L33:0  INS_6_POS
  L192:1  BOT_LAST_TIME  "rtc bot belt previous movement event time"
  L192:2  BOT_CYCLE_TIME  "rtc bot belt time between events"
  L192:7  FROM_REAL  "distance from real part signal at optic location"
  L192:8  FROM_TRACKED  "distance from tracked part signal at optic location"
  L192:16  TOP_LAST_TIME  "rtc top belt previous movement event time"
  L192:17  TOP_CYCLE_TIME  "rtc top belt time between events"
  L199:5  ACQTM51
  L199:6  ACQTM52
  L199:7  ACQTM53
  L199:9  "ones"
  L199:10  "billions"
  L199:13  DUMP_LONG
  L199:15  ACQTM11
  L199:16  ACQTM12
  L199:17  ACQTM13
  L199:20  RESULTTM1
  L199:22  CLEARTIME5COUNT
  L199:23  CLEARTIME6COUNT
  L199:24  ACQTM61
  L199:25  ACQTM62
  L199:26  ACQTM63
  L199:27  TMSINCETRIG1
  L199:29  TMSINCETRIG5
  L199:30  TMSINCETRIG6
  L199:31  CLEARTIME1COUNT
  L199:32  RESULTTM5
  L199:33  RESULTTM6
  L199:34  MAXACQTM1
  L199:36  MAXACQTM6
  N7  
  N101:2  I3_TRIG_LOC
  N101:3  I4_TRIG_LOC
  O:0.0/1  "spare"
  O:0.0/11  "Spare"
  O:0.0/12  "not used"
  O:0.0/13  "not used"
  O:0.0/14  "not used"
  O:0.0/15  "not used"
  O:0.1  "not used"
  O:0.2  "not used"
  O:0.3  "not used"
  O:0.5  "spare analog output"
  O:3.0/0  "spare"
  O:3.0/2  "spare"
  O:3.0/3  "light curtain range selection /* needed? */"
  O:3.0/7  "door unlocks on CE models"
  O:3.0/8  "Light?"
  O:3.0/9  NUT_HOPPER  "Nut Hopper Enable"
  O:3.0/11  NUT_FEEDER_AIR  "Nut Feeder Bowl Air Enable"
  PFILE:6  "check for part jams"
  PFILE:10  "Bottom belt HSC"
  PFILE:12  "Top belt HSC"
  Q2:55  END_OF_MAIN
  Q5:94  END_OF_BELTS
  T20:0  "Trigger On Time"
  U:9  "slow data"
  U:24  "check skipped fail rate"
  U:28  "faults"
  U:29  "speed"
  U:30  "count"
  U:31  "rate calc"
  U:32  "boxer"
  U:33  "bulk pack"
  U:34  "customer boxing unit signals"
  U:35  "cleanup"

COMMENTS NOT ATTACHED TO A CURRENT RUNG
  R6:2: B41 is the top good 3 file
  R6:6/DN: B35 is the top NG file
  R6:10/DN: B37 is the top good 1 file
  R6:11/DN: B39 is the top good 2 file
  R6:0: B36 is the bottom GOOD file
  R6:10: B37 is the top good 1 file
  R6:6: B35 is the top NG file
  R6:4: B34 is the bottom NG file

REVISION NOTES
  13: updated count reset
  14: added io moduals
  15: multiple steps toward new hmi integration
  21: test
  27: fix error if bulk pack and no boxing fallout were on

DATA TABLE (non-zero values as saved)
DATA B3
% B3:0 % 0X8822 0X0141 0X5001 0XA109 0XEC97 0X3540 0X0C30 0X0421 0X3F80 0X2550
% B3:10 % 0X21E0 0X40C6 0X4000 0X10D4 0X0011 0X0000 0X0000 0X0000 0X0000 0X0000
% B3:50 % 0X0001 0X0000 0X0000 0X0000 0X0000 0X0000 0X0000 0X0000 0X0000 0X0000
DATA T4
% .PRE .ACC %
% T4:1 % 150 152
% T4:2 % 400 0
% T4:3 % 125 0
% T4:4 % 1000 0
% T4:5 % 5 5
% T4:6 % 10 32766
% T4:7 % 150 0
% T4:8 % 20 2
% T4:9 % 50 24
% T4:10 % 200 200
% T4:11 % 111 0
% T4:12 % 40 42
% T4:13 % 250 0
% T4:14 % 666 0
% T4:15 % 1000 1001
% T4:16 % 400 0
% T4:17 % 100 57
% T4:18 % 5 0
% T4:19 % 300 0
% T4:20 % 200 0
% T4:21 % 200 0
% T4:22 % 200 0
% T4:23 % 250 0
% T4:24 % 666 0
% T4:25 % 666 0
% T4:26 % 666 0
% T4:27 % 250 0
% T4:28 % 250 0
% T4:29 % 10000 0
% T4:30 % 333 0
% T4:31 % 125 0
% T4:32 % 300 277
% T4:33 % 222 166
% T4:34 % 1111 0
% T4:35 % 23 0
DATA C5
% .PRE .ACC %
% C5:0 % 32766 0
DATA R6
% .LEN .POS %
% R6:0 % 1400 0
% R6:1 % 16 0
% R6:2 % 1050 0
% R6:3 % 1050 0
% R6:4 % 1400 0
% R6:5 % 1250 0
% R6:6 % 1713 0
% R6:7 % 16 0
% R6:8 % 1024 0
% R6:9 % 3 0
% R6:10 % 1713 0
% R6:11 % 1050 0
% R6:12 % 10 0
% R6:13 % 10 0
% R6:14 % 10 0
% R6:15 % 10 0
% R6:16 % 1713 0
% R6:17 % 1713 0
% R6:18 % 1050 0
% R6:19 % 10 0
DATA N7
% N7:0 % 32767 6 938 194 3 0 0 0 500 43
% N7:10 % 1 43 0 8 22 22 1000 2000 50 100
% N7:20 % 0 1329 16 2000 0 48 0 0 0 250
% N7:30 % 666 32767 150 0 728 1317 82 11 1 10
% N7:40 % 1 38 1 37 187 1266 32767 1266 0 0
% N7:50 % 16 16 0 16 17 712 0 32767 0 3
% N7:60 % 1713 1713 1050 937 1034 1024 4999 5 400 400
% N7:70 % 100 200 300 400 90 190 290 390 25992 32767
% N7:80 % 0 0 1346 1352 1392 1402 84 27 0 0
% N7:90 % 2011 4 4 12 1 84 27 222 222 12
% N7:100 % 1003 90 110 100 175 25 0 0 0 0
% N7:190 % -128 27477 27605 32767 0 0 0 0 0 0
DATA F8
% F8:0 % 6
DATA L13
% L13:0 % 208468 519392 0 229384 718622
% L13:5 % 113540 166063 146116 673920 123873
% L13:10 % 132269 40154 74267 15 90
% L13:15 % 847054163 -2147483648 2147483647 2147483647 82058
% L13:20 % 469867010 -1285684965 777 62053 100
% L13:25 % 91423 19753 -340487 0 845055429
% L13:30 % 1997911 113540 1020000 846295376 1444
% L13:35 % 0 46 99 -722056871 -722056831
% L13:40 % 16256 1000000000 1000000 846295200 846939870
% L13:45 % 846423123 40 0 176 469829770
% L13:50 % 114337 111825 145888338 130 0
% L13:55 % 631084 130 15196 82392030 82395466
% L13:60 % 7723 2085602 0 600 15
% L13:65 % 100 1500 -722055583 -722055545 2
% L13:70 % 322164536 139 8 1625600 469829770
% L13:75 % 59 30 100 919373699 1
% L13:80 % 557730 74 74 40 1519592
% L13:85 % 210337 168 167 0 114360
% L13:90 % 631107 3 253667 5 846939922
% L13:95 % 99 132 0 846423171 199461
% L13:100 % 100 7 -2147483648 1111 337
% L13:105 % 199461 568360 469783569 4633 469783558
% L13:110 % 11 33 66 -1285935441 -1285895295
% L13:115 % -1285895287 8 4 -1285895291 1000
% L13:120 % 105738436 2987 99 115 303
% L13:125 % 0 322164536 -8733 3276500 250501
% L13:130 % 33 66 0 249 -249
% L13:135 % 0 500 210347 1000 0
% L13:140 % 36696000 36696000 36 50 50
% L13:145 % 111826 5 131 5 20
% L13:150 % 12 20 380641 -380641 40154
% L13:155 % 1 -8 36696000 1 4589052
% L13:160 % 16 52 48 1220 45
% L13:165 % -1285722992 -1285894889 -1285722992 -1285894889 6706
% L13:170 % 12817 305 8978 700 200
% L13:175 % 4 4 42 23 38
% L13:180 % -722038264 57 50833 1000000 167000000
% L13:185 % 0 0 -722038314 57 50918
% L13:190 % 168000000 0 0 0 0
% L13:205 % 0 0 0 518736 541928
DATA L19
% L19:0 % 845055429 845062934 845070342 845077727 845085012
% L19:5 % 845092504 845099769 845107067 845114280 845121070
% L19:10 % 845128533 845135356 845142733 845149565 845157008
% L19:15 % 846412950 846421927 0 0 0
DATA L20
% L20:0 % 846914206 846914510 846914816 846915122 846915429
% L20:5 % 846915734 846916038 846916344 846916648 846916953
% L20:10 % 846917258 846917564 846917869 846918175 846918479
% L20:15 % 846918783 846919088 846919394 846919701 846920008
% L20:20 % 846920311 846920617 846920922 846921228 846921532
% L20:25 % 846921838 846922144 846922449 846922755 846923062
% L20:30 % 846923368 846923672 846923978 846924285 846924590
% L20:35 % 846924896 846925202 846925509 846925813 846926119
% L20:40 % 846926427 846926733 846927040 846927345 846927650
% L20:45 % 846927955 846928261 846928567 846928871 846929177
% L20:50 % 846929482 846929788 846930094 846930400 846930705
% L20:55 % 846931012 846931318 846931624 846931930 846932235
% L20:60 % 846932540 846932846 846933151 846933457 846933763
% L20:65 % 846934068 846934375 846934679 846934986 846935292
% L20:70 % 846935599 846935904 846936209 846936515 846936820
% L20:75 % 846937126 846937431 846937736 846938041 846938346
% L20:80 % 846938650 846938955 846939259 846939565 846939870
% L20:85 % 846909621 846909929 846910235 846910540 846910846
% L20:90 % 846911151 846911456 846911760 846912065 846912370
% L20:95 % 846912677 846912984 846913289 846913595 846913900
DATA L21
% L21:0 % -1285731528 -1285731427 -1285731325 -1285731223 -1285731121
% L21:5 % -1285731020 -1285730919 -1285730817 -1285730716 -1285730614
% L21:10 % -1285730513 -1285730411 -1285730310 -1285730208 -1285730107
% L21:15 % -1285730006 -1285729904 -1285729803 -1285729701 -1285729598
% L21:20 % -1285729498 -1285729396 -1285729295 -1285729193 -1285729092
% L21:25 % -1285728990 -1285728888 -1285728786 -1285728685 -1285728583
% L21:30 % -1285728481 -1285728380 -1285728278 -1285728176 -1285728074
% L21:35 % -1285727972 -1285727871 -1285727769 -1285727668 -1285727566
% L21:40 % -1285727463 -1285727362 -1285727260 -1285727158 -1285727056
% L21:45 % -1285726955 -1285726853 -1285726751 -1285726650 -1285726549
% L21:50 % -1285726447 -1285726345 -1285726244 -1285726142 -1285726040
% L21:55 % -1285725938 -1285725836 -1285725735 -1285725633 -1285725531
% L21:60 % -1285725430 -1285725328 -1285725227 -1285725125 -1285725023
% L21:65 % -1285724922 -1285724819 -1285724718 -1285724616 -1285724514
% L21:70 % -1285724412 -1285724311 -1285724209 -1285724108 -1285724006
% L21:75 % -1285723905 -1285723803 -1285723702 -1285723600 -1285723499
% L21:80 % -1285723398 -1285723296 -1285723195 -1285723093 -1285722992
% L21:85 % -1285733053 -1285732951 -1285732849 -1285732747 -1285732646
% L21:90 % -1285732544 -1285732442 -1285732341 -1285732240 -1285732138
% L21:95 % -1285732036 -1285731934 -1285731833 -1285731731 -1285731630
DATA L22
% L22:0 % 845049526 845056626 845064129 845071539 845078923
% L22:5 % 845086208 845093699 845100966 845108262 845115476
% L22:10 % 845122265 845129729 845136552 845143930 845150760
% L22:15 % 845158203 846293307 846293537 846293769 846294001
% L22:20 % 846294230 846294459 846294689 846294920 846295147
% L22:25 % 846295379 846414145 846423123 843151733 843151961
% L22:30 % 843152189 843152417 843152644 843152871 843745038
% L22:35 % 843797842 843845258 843982696 844020075 844041926
% L22:40 % 844058091 844077200 844989306 844996663 845003856
% L22:45 % 845013515 845020858 845027993 845035009 845042281
DATA L23
% L23:0 % -1286351836 -1286349474 -1286346977 -1286344512 -1286342056
% L23:5 % -1286339632 -1286337141 -1286334724 -1286332297 -1286329897
% L23:10 % -1286327639 -1286325156 -1286322886 -1286320432 -1286318160
% L23:15 % -1286315684 -1285938073 -1285937996 -1285937919 -1285937842
% L23:20 % -1285937766 -1285937690 -1285937613 -1285937536 -1285937461
% L23:25 % -1285937384 -1285897876 -1285894889 -1286797739 -1286797739
% L23:30 % -1286797739 -1286797739 -1286797739 -1286797739 -1286785787
% L23:35 % -1286768219 -1286752447 -1286706724 -1286694291 -1286687021
% L23:40 % -1286681644 -1286675289 -1286371869 -1286369421 -1286367029
% L23:45 % -1286363816 -1286361373 -1286358999 -1286356665 -1286354246
DATA L30
% L30:0 % 846293877 846294010 846294140 846294272 846294404
% L30:5 % 846294537 846294670 846294802 846294934 846295067
% L30:10 % 846295200 846295332 769495134 769507325 769518683
% L30:15 % 769530479 769542633 769553775 769565037 843150665
% L30:20 % 843150795 843150924 843151054 843151184 843151315
% L30:25 % 843151446 843151575 843151704 843151835 843151963
% L30:30 % 843152093 843152223 843152352 843152483 843152614
% L30:35 % 843152746 843718651 843725666 843737833 843766618
% L30:40 % 843778510 843790666 843824106 843838046 846293087
% L30:45 % 846293218 846293350 846293482 846293615 846293746
DATA L31
% L31:0 % 469829330 469829375 469829418 469829461 469829505
% L31:5 % 469829550 469829594 469829638 469829681 469829726
% L31:10 % 469829770 469829814 469350498 469354555 469358338
% L31:15 % 469362254 469366300 469370009 469373757 469740804
% L31:20 % 469740804 469740804 469740804 469740804 469740804
% L31:25 % 469740804 469740804 469740804 469740804 469740804
% L31:30 % 469740804 469740804 469740804 469740804 469740804
% L31:35 % 469740804 469743983 469746308 469750358 469759935
% L31:40 % 469763894 469767929 469779058 469783691 469829068
% L31:45 % 469829111 469829156 469829200 469829243 469829286
DATA L32
% L32:0 % 145888338 145887663 145888001 -541039302 -541039076
% L32:5 % -541038851 -541038626 -541038400 -541038175 -541037948
% L32:10 % 227357062 227357287 227357512 227357738 227357963
% L32:15 % 227358188 227358414 227358639 227358864 919354909
% L32:20 % 919355134 919355360 919355585 919355810 919356036
% L32:25 % 919356261 919356487 919356711 919356936 919373560
% L32:30 % -103475746 -103475626 -103475288 -614834856 -614834631
% L32:35 % -614834406 -614834180 -614833955 -614833730 -614833504
% L32:40 % -614833279 -614833054 -614832829 -614832603 -614832379
% L32:45 % -614832152 -614831927 -614831702 -614831476 -614831251
DATA L33
% L33:0 % 427902972 427902972 427902972 322161012 322161012
% L33:5 % 322161012 322161012 322161012 322161012 322161012
% L33:10 % 322161335 322161335 322161335 322161335 322161335
% L33:15 % 322161335 322161335 322161335 322161335 322161354
% L33:20 % 322161354 322161354 322161354 322161354 322161354
% L33:25 % 322161354 322161354 322161354 322161354 322164536
% L33:30 % 427902972 427902972 427902972 322161011 322161011
% L33:35 % 322161011 322161011 322161011 322161011 322161011
% L33:40 % 322161011 322161011 322161011 322161011 322161011
% L33:45 % 322161011 322161011 322161011 322161011 322161011
DATA B35
% B35:110 % 0X0000 0X0000 0X0200 0X0000 0X0000 0X0000 0X0000 0X0000 0X0000 0X0000
DATA B37
% B37:0 % 0X0000 0X0000 0X2000 0X0000 0X0000 0X0000 0X0000 0X0000 0X0000 0X0000
DATA B40
% B40:0 % 0XAAAA
DATA B41
% B41:50 % 0X0000 0X0000 0X0000 0X0000 0X0FF0 0X0000 0X0000 0X0000 0XBFC0 0XA586
DATA B100
% B100:0 % 0X2780 0X18A0 0X0004 0X0000 0X0000 0X0000 0X0000 0X0000 0X0000 0X0000
DATA N101
% N101:0 % 128 646 0 0 1294 100 934 1200 1200 1326
% N101:10 % 1336 1602 10 15727 778 17365 1566 125 333 125
% N101:20 % 1000 500 400 0 1 0 222 300 0 0
DATA L102
% L102:0 % 40 8 3272 3305 3300
% L102:5 % 3300 1 0 0 0
% L102:10 % 0 1 0 0 253667
% L102:15 % 0 30 18 30 19
% L102:20 % 388 7 32165 2 52
% L102:25 % 176 0 1 32613 1
% L102:30 % 139 0 -1022849445 166833 -6372355
% L102:35 % 446 50000 0 999999 48
% L102:40 % 0 2 22080 0 0
